PROGRAM AdsClient_1
VAR_OUTPUT
	ServerPrgName		: STRING;
	ServerNetId			: STRING; 	(* Server AmsNetId *)
	ServerPort 			: UINT;		(* Server port number *)
	
	LocalPrgName		: STRING;// := 'AREA_2';
	LocalNetId			: STRING;
	LocalPort			: UINT;// := 851;

	bBusy				: BOOL;
	err					: BOOL;
	errId				: UDINT;
	
	socketReady			: BOOL;
	
	remoteAccessPrefix	: STRING := 'AdsServer.area[2].';
END_VAR
VAR
	setupTimer 			: TON;
	
	handle				: AdsHandle_1;
	numHandles 			: INT(0..maxHandles);
	
	setupStep 			: (SET_LOCAL_ENDPOINT, CLOSE_CONNECTIONS, SEND_CONNECTION_DATA, RECEIVE_SERVER_DATA, FINISH_SETUP);
	
	fbGetLocalAmsNetId	: FB_GetLocalAmsNetId;
END_VAR
VAR CONSTANT
	maxHandles			: INT := 6;
END_VAR

socketReady := setup();

IF NOT socketReady THEN //setup after initialization
	RETURN;
END_IF
	
handle(
	RemotePrgName=> ServerPrgName, 
	RemoteNetId=> ServerNetId, 
	RemotePort=> ServerPort, 
	LocalPrgName=> LocalPrgName, 
	LocalNetId=> LocalNetId, 
	LocalPort=> LocalPort, 
	remoteAccessPrefix=> , 
	busy=> , 
	error=> , 
	errorId=> , 
	receiveBuffer=> , 
	receiveStruct=> );

METHOD fetchData : BOOL
VAR_IN_OUT
	receiverStruct : AdsData;
END_VAR
VAR
	emptyData : AdsData;
END_VAR
receiverStruct := handle.receiveStruct;

fetchData := MEMCMP(ADR(receiverStruct), ADR(emptyData), SIZEOF(AdsData)) <> 0; //returns false if no data

handle.clearBuffer();
END_METHOD

METHOD PROTECTED findHandle : REFERENCE TO AdsHandle
VAR_INPUT
	remotePrgName : STRING;
END_VAR
IF handle.getHandlerName() = remotePrgName THEN
	findHandle REF= handle;
	RETURN;
END_IF
END_METHOD

METHOD queueData : BOOL
VAR_INPUT
	data : REFERENCE TO AdsData;
END_VAR
handle.queueData(data);
END_METHOD

METHOD PROTECTED read : BOOL
VAR_INPUT
	remotePrgName : STRING;
	symbol : STRING;
	buffer : PVOID;
	symbolSize : UDINT;
END_VAR
VAR
	targetHandler : REFERENCE TO AdsHandle;
END_VAR
targetHandler REF= findHandle(remotePrgName);

IF __ISVALIDREF(targetHandler) THEN
	targetHandler.read(symbol, buffer, symbolSize);
END_IF
END_METHOD

METHOD PROTECTED send : BOOL
VAR_INPUT
	data : PVOID;
	dataSize : UDINT;
END_VAR
write(CONCAT(remoteAccessPrefix, 'genericBuffer'), data, dataSize);
END_METHOD

METHOD PROTECTED setup : BOOL
VAR
	pass : BOOL;
END_VAR
fbGetLocalAmsNetId(
	bExecute:= , 
	tTimeOut:= , 
	bBusy=> , 
	bError=> , 
	nErrId=> , 
	AddrString=> LocalNetId, 
	AddrBytes=> );
fbGetLocalAmsNetId.bExecute := NOT fbGetLocalAmsNetId.bExecute;

LocalPrgName := 'AREA_2';
LocalPort := 851;

handle.setup();




(*
IF
	localPrgName <> '' AND
	localNetId <> '' AND localNetId <> '0.0.0.0.0.0' AND
	localPort <> 0
THEN
	fbGetLocalAmsNetId.bExecute := FALSE;
	handle.open(localPrgName, localNetId, localPort);
	
	setupStep := CLOSE_CONNECTIONS;
END_IF

handle.setup();
*)
(*
CASE setupStep OF
	SET_LOCAL_ENDPOINT:
		localPrgName := 'AREA_2';
		localPort := 851;
		
		fbGetLocalAmsNetId(
			bExecute:= , 
			tTimeOut:= , 
			bBusy=> , 
			bError=> , 
			nErrId=> , 
			AddrString=> localNetId, 
			AddrBytes=> );
		fbGetLocalAmsNetId.bExecute := NOT fbGetLocalAmsNetId.bExecute;	
		
		IF
			localPrgName <> '' AND
			localNetId <> '' AND localNetId <> '0.0.0.0.0.0' OR
			localPort <> 0
		THEN
			fbGetLocalAmsNetId.bExecute := FALSE;
			handle.open(localPrgName, localNetId, localPort);
			
			setupStep := CLOSE_CONNECTIONS;
		END_IF
		
	CLOSE_CONNECTIONS:
		handle.close();
		setupStep := SEND_CONNECTION_DATA;
		
	SEND_CONNECTION_DATA:
		CASE adsCtr OF
			0:
				pass := handle.write(
					symbol:= 'AdsServer.handle[1].remotePrgName',
					data:= ADR(localPrgName),
					dataSize:= SIZEOF(localPrgName));
			
			1:
				pass := handle.write(
					symbol:= 'AdsServer.handle[1].remoteNetId',
					data:= ADR(localNetId),
					dataSize:= SIZEOF(localNetId));
			
			2:
				pass := handle.write(
					symbol:= 'AdsServer.handle[1].remotePort',
					data:= ADR(localPort),
					dataSize:= SIZEOF(localPort));
			
			3:
				adsCtr := 0;
				setupStep := RECEIVE_SERVER_DATA;
				RETURN;
			
		END_CASE
		
		IF pass THEN
			adsCtr := adsCtr + 1;
		END_IF
		
	RECEIVE_SERVER_DATA:
		CASE adsCtr OF
			0:
				pass := handle.read(
					symbol:= 'AdsServer.handle[2].socket.localPrgName', 
					buffer:= ADR(handle.socket.remotePrgName), 
					symbolSize:= SIZEOF(handle.socket.remotePrgName));
			
			1:
				pass := handle.read(
					symbol:= 'AdsServer.handle[2].socket.localNetId', 
					buffer:= ADR(handle.socket.remoteNetId), 
					symbolSize:= SIZEOF(handle.socket.remoteNetId));
			
			2:
				pass := handle.read(
					symbol:= 'AdsServer.handle[2].socket.localPort', 
					buffer:= ADR(handle.socket.remotePort), 
					symbolSize:= SIZEOF(handle.socket.remotePort));
			
			3:
				adsCtr := 0;
				setupStep := FINISH_SETUP;
				RETURN;
			
		END_CASE
		
		IF pass THEN
			adsCtr := adsCtr + 1;
		END_IF
			
	FINISH_SETUP:
		setup := TRUE;
		RETURN;
END_CASE
*)
END_METHOD

METHOD PROTECTED write : BOOL
VAR
	remotePrgName : STRING := handle.socket.remotePrgName;
END_VAR
VAR_INPUT
	symbol : STRING;
	data : PVOID;
	dataSize : UDINT;
END_VAR
VAR
	targetHandle : REFERENCE TO AdsHandle;
END_VAR
targetHandle REF= findHandle(remotePrgName);

IF __ISVALIDREF(targetHandle) THEN
	targetHandle.write(symbol, data, dataSize);
END_IF
END_METHOD

END_PROGRAM

(* stored: Version 1.1.0.1, ProductVersion 3.1.4024.11
   POU AdsClient_1: Id {e7dcd06c-b780-4180-89ff-e14ebb81dac3}, SpecialFunc None
   Folder ADS: Id {51440617-69f3-466b-9900-c9c81e97d18f}
   Method fetchData: Id {054516b2-9a3c-45c9-af8f-a7b1ab7efee9}
   Method findHandle: Id {9977c594-58ba-4387-b51c-44f23c733f0d}
   Method queueData: Id {4a072abd-19ca-42bf-8b6d-164efc13b966}
   Method read: Id {5181b838-db8b-4a54-8427-cf976e4f76dc}
   Method send: Id {b2751e23-9abf-44ce-8110-054559037076}
   Method setup: Id {ebeacf4a-f5a0-469b-a395-4778f5b31d6c}
   Method write: Id {07e8464b-5ad2-4dc1-8ecd-5f2ae5317a8c} *)
